ABB RobotStudio station: Tp2_20201212-063412.rsstn

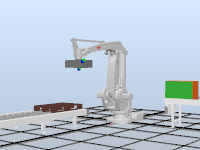
Station Tp2 (saved by RobotStudio 20.1.8982.0)
Layout (positions relative to the parent item):
  - transporteCajas [part, from Equipment\Conveyor Guide 400.rslib] at (0, 1500, 0) mm, rotated rx 0 ry 0 rz 90 deg
  - Euro Pallet [graphiccomponentgroup, from Equipment\Euro Pallet.rslib] at (1000, -1425, 435) mm
    - Body 1 [part, from Equipment\Euro Pallet.rslib]
  - transportePallets [part, from Equipment\Conveyor 950 4000 h2.rslib] at (1000, -1500, 0) mm
  - caja [part] at (-200, 1500, 770) mm
  - IRB660_180_315__01_2 [mechanism, from Robots\IRB660_180_315__01.rslib] at (0, 0, 0) mm; joint values [0, 0, 0, 0] (rad or m)
  - ventosa_tool [mechanism] at (1910, 0, 1833) mm, rotated rx 180 ry 0 rz 180 deg
      TCP ventosa_tool at (0, 0, 200) mm
      links: ventosa
  - topePallet [frame] at (1000, -1025, 435) mm
  - basePallet [frame] at (1000, -1025, 435) mm
  - topeCajas [frame] at (-200, 1500, 770) mm
Attachment: Euro Pallet is attached to transportePallets
Attachment: basePallet is attached to Euro Pallet
Attachment: topePallet is attached to transportePallets
Attachment: topeCajas is attached to transporteCajas
Attachment: ventosa_tool is attached to IRB660_180_315__01_2 / Link6
Targets, tools, work objects and paths stored in the station, written as RAPID:
! task (no controller)
MODULE CalibData
  PERS tooldata ventosa_tool:=[TRUE,[[0,0,200],[1,0,0,0]],[1,[0,0,1],[1,0,0,0],0,0,0]];
ENDMODULE

